DATA_BLOCK "DB_IN"	// DB 111
AUTHOR : M.Kögel
VERSION : 0.1
  STRUCT
   EMX_SPINDLE_RUN : BOOL ;	//Spindel läuft
   EMX_PROGRAM_RUN : BOOL ;	//Programm läuft
   EMX_FEED_HOLD : BOOL ;	//Vorschuboverride = 0 oder Voschub Stopp
   EMX_WARNING : BOOL ;	//Warnmeldung
   EMX_ERROR : BOOL ;	//Fehlermeldung
   EMX_FUNCTION_M20 : BOOL ;	//Funktion M20/M190
   EMX_PROGRAM_HALT : BOOL ;	//programmierter Halt "M00"
   EMX_AXIS_MOVE : BOOL ;	//mindestens eine Hauptachse in Bewegung
   EMX_MANUAL_MODE : BOOL ;	//Betriebsart Manuell
   EMX_TEACH_MODE : BOOL ;	//Betriebsart Teach
   EMX_SINGLE_MODE : BOOL ;	//Betriebsart Einzelsatz
   EMX_AUTO_MODE : BOOL ;	//Betriebsart Auto
   EMX_CYCLE_START : BOOL ;	//Zyklus Start (Starttaste - grün)
   EMX_MACHINE_ON : BOOL ;	//Maschine ist eingeschaltet (KEIN Not-Aus)
   EMX_NC_READY2RUN : BOOL ;	//NC-Betriebsbereit
   EMX_PROGRAM_END : BOOL ;	//Programm Ende
   EMB_PALLET_NUMBER : BYTE ;	//Nummer der Palette im Arbeitsraum
   EMX_PC_ACTIVE : BOOL ;	//Palettenwechsel aktiv
   EMX_SUS_DOOR_LOCKED : BOOL ;	//Rüstplatztüre(n) geschlossen und verriegelt
   EMX_PALLET_ON_SUS : BOOL ;	//Palette am Rüstplatz vorhanden
   EMX_ERROR_PULSE : BOOL ;	//Impuls von 1sec bei jeder Fehlermeldung
   EMX_PC_RELEASED : BOOL ;	//Freigabe für Palettenwechsel ist aktiv
   EMX_PC_PROCESS_END : BOOL ;	//Palettenwechsel beendet (nachdem Palette geklemmt)
   EMX_SUS_DOOR_CLOSED : BOOL ;	//Rüstplatztüre(n) geschlossen
   EMX_PC_CHANGE_POS : BOOL ;	//Maschinenpalette auf Übergabeposition (vor Hubbewegung)
   EMX_COOLANT_M8 : BOOL ;	//äußere Kühlschmierstoffzufuhr
   EMX_COOLANT_M7 : BOOL ;	//innere Kühlschmierstoffzufuhr
   EMX_FLUSH_PALLET : BOOL ;	//Spülung Palettenträger aktiv
   EMX_COOLANT_BACKFLOW : BOOL ;	//Förderpumpe Sammelbehälter (Rückförderung aus Maschine)
   EMX_COOLANT_LACK : BOOL ;	//Vorwarnung Kühlschmierstoffmangel
   EMX_COOLANT_MINLEVEL : BOOL ;	//Kühlschmierstoffanlage Füllstand minimum
   EMX_LUBRICAT_MINLEVEL : BOOL ;	//Zentralschmierung Füllstand minimum
   EMX_MQL_MINLEVEL : BOOL ;	//Minimalmengenschmierung Füllstand minimum
   EMX_HYDR_MINLEVEL : BOOL ;	//Hydraulikaggregat Werkzeugmaschine Füllstand minimum
   EMX_HYDRCHUCK_MINLEVEL : BOOL ;	//Hydraulikaggregat Spannhydraulik Füllstand minimum
   frei52 : BOOL ;
   frei53 : BOOL ;
   frei54 : BOOL ;
   frei55 : BOOL ;
   frei56 : BOOL ;
   frei57 : BOOL ;
   EMX_FEEDRATE_X : BOOL ;	//Vorschuboverride größer Wert "X"
   EMX_TOOL_LIFE : BOOL ;	//Standzeit des aktuellen Werkzeuges abgelaufen
   EMX_TOOL_CHANGE : BOOL ;	//Werkzeugwechsel aktiv
   EMX_MQL_ACTIVE : BOOL ;	//Minimalmengenschmierung aktiv (M34/M35)
   EMX_TOOL_LIFE_PREWARN : BOOL ;	//Die Standzeit des aktuellen Werkzeuges hat die Vorwarngrenze überschritten
   EMX_MAINTENANCE_REMIN : BOOL ;	//Wartungsaufruf (gemäß Betriebsanleitung; bei Maschinenfunktion (Dauer =250h)
   EMX_LUBRICAT_ACTIVE : BOOL ;	//High-Pegel, wenn die Zentral- (Maschinen)schmierung aktiviert ist
   ImxToolBreakage : BOOL ;	//Werkzeugbruch, welcher ein Stop auslöst
   EMX_ALARM_RESET : BOOL ;	//Meldung quittieren
   EMX_WORKROOM_DOOR : BOOL ;	//Arbeitsraumtüre(n) der Werkzeugmaschine geschlossen und verriegelt
   EMX_ZPS_RELEASE_EXT : BOOL ;	//Nullpunktspannsystem lösen (von extern)
   EMX_FIXTURE_ON_SUS : BOOL ;	//Palette mit (externem) Spannsystem auf Rüstplatz (MAS, RS4)
   frei74 : BOOL ;
   EMX_UNLOCK_FIXTURE : BOOL ;	//Freigabe für Spannvorrichtung lösen (Handling)
   frei76 : BOOL ;
   frei77 : BOOL ;
   EMX_OPERATING_MODE2 : BOOL ;	//Betriebsart_2 aktiv (Einrichtbetrieb)
   EMX_OPERATING_MODE3 : BOOL ;	//Betriebsart_3 aktiv (manueller Eingriff)
   EMX_OPERATING_MODE4 : BOOL ;	//Betriebsart_4 aktiv (erweiterter manueller Eingriff )
   EMX_AXIS_STANDSTILL : BOOL ;	//Achsenstillstand (Arbeitsraum) X/Y/Z/S/A/B/C-Achse
   EMX_STROBE_FUNCTION1 : BOOL ;	//Zustandswechsel an Funktionsaufruf (EMW_FUNCTION1)
   EMX_TURNTABLE_RUN : BOOL ;	//Fräs-Drehtisch läuft im Drehbetrieb
   frei86 : BOOL ;
   frei87 : BOOL ;
   EMX_SUS_PRESSURELESS : BOOL ;	//Medienübergabe am Rüstplatz (des PW oder des Rundspeichers) drucklos
   EMX_SUS_COUPLED : BOOL ;	//Andockeinheit (Medienversorgung) am Rüstplatz ausgefahren (gekuppelt)
   EMX_SUS_DOOR_OPENED : BOOL ;	//Rüstplatztüre des Speichersystem (z.B. RS4) vollständig geöffnet
   ImxOpenSusDoor : BOOL ;	//Rüstplatztüre(n) öffnen
   ImxCloseSusDoor : BOOL ;	//Rüstplatztüre(n) schließen
   frei95 : BOOL ;
   frei96 : BOOL ;
   frei97 : BOOL ;
   EMW_PARAMETER_1 : WORD ;	//Konfiguration über Maschinenparameter_1
   EMW_PARAMETER_2 : WORD ;	//Konfiguration über Maschinenparameter_2
   EMW_PARAMETER_3 : WORD ;	//Konfiguration über Maschinenparameter_3
   EMW_PARAMETER_4 : WORD ;	//Konfiguration über Maschinenparameter_4
   EMB_FEEDRATE : BYTE ;	//Stellung(Position) des Vorschubpotentiometers(Override)
   EMB_RAPID_VELOCITY : BYTE ;	//Stellung des Eilgangspotentiometers (Override)
   EMW_FUNCTION1 : WORD ;	//Funktionsaufruf durch Teileprogramm
   ImxDataRoutingBit0 : BOOL ;	//RANGIERER EINGANG BIT0
   ImxDataRoutingBit1 : BOOL ;	//RANGIERER EINGANG BIT1
   ImxDataRoutingBit2 : BOOL ;	//RANGIERER EINGANG BIT2
   ImxDataRoutingBit3 : BOOL ;	//RANGIERER EINGANG BIT3
   ImxDataRoutingBit4 : BOOL ;	//RANGIERER EINGANG BIT4
   ImxDataRoutingBit5 : BOOL ;	//RANGIERER EINGANG BIT5
   ImxDataRoutingBit6 : BOOL ;	//RANGIERER EINGANG BIT6
   ImxDataRoutingBit7 : BOOL ;	//RANGIERER EINGANG BIT7
   ImxDataRoutingBit8 : BOOL ;	//RANGIERER EINGANG BIT8
   ImxDataRoutingBit9 : BOOL ;	//RANGIERER EINGANG BIT9
   ImxDataRoutingBit10 : BOOL ;	//RANGIERER EINGANG BIT10
   ImxDataRoutingBit11 : BOOL ;	//RANGIERER EINGANG BIT11
   ImxDataRoutingBit12 : BOOL ;	//RANGIERER EINGANG BIT12
   ImxDataRoutingBit13 : BOOL ;	//RANGIERER EINGANG BIT13
   ImxDataRoutingBit14 : BOOL ;	//RANGIERER EINGANG BIT14
   ImxDataRoutingBit15 : BOOL ;	//RANGIERER EINGANG BIT15
   ImbSpindleOverride : BYTE ;	//Stellung des Spindeldrehzahlkorrekturschalters
  END_STRUCT ;	
BEGIN
END_DATA_BLOCK

DATA_BLOCK "DB_OUT"	// DB 112
AUTHOR : APetz
VERSION : 0.1
  STRUCT
   AMX_FEED_STOP : BOOL ;	//Vorschub Stopp  (mit Fehlermeldung)
   AMX_FEED_HOLD_CYCLE : BOOL ;	//Vorschub Halt (gilt nicht bei Eilgang-G00) mit Warnung
   AMX_SPINDLE_FEED_STOP : BOOL ;	//Spindel und Vorschub Stopp (mit Fehlermeldung)
   AMX_SPINDLE_FEED_STOP_P : BOOL ;	//Spindel und Vorschub Stopp nach abgearbeitetem Satz (mit Fehlermeldung)
   AMX_EMERGENCY_STOP : BOOL ;	//Not-Aus
   AMX_EMERGENCY_STOP_P : BOOL ;	//Not-Aus nach abgearbeitetem Satz
   AMX_LUBRICATION_LEVEL : BOOL ;	//Füllstandsüberwachung Schmieraggregat -> Warnmeldung
   AMX_SPINDLE_FEED_STOP_G0 : BOOL ;	//Spindel und Vorschub Stopp beim nächstem G0
   AMX_PC_RELEASE : BOOL ;	//Freigabe Palettenwechsler (Taste)
   AMX_PC_LOCK : BOOL ;	//Palettenwechsler sperren
   AMX_PC_ENABLE : BOOL ;	//Palettenwechselablauf freigeben
   AMX_STACKER_LOCK : BOOL ;	//Fahraufträge des Speichersystems vom und zum Rüstplatz sperren
   frei14 : BOOL ;
   frei15 : BOOL ;
   frei16 : BOOL ;
   frei17 : BOOL ;
   AMX_ERROR_KSS : BOOL ;	//Fehlermeldung Späneförderer/Kühlmittel
   AMX_FLOW_CONTROL_M7 : BOOL ;	//Kühlmitteldurchfluss im Kühlschmierstoff-Hochdruckkreis vorhanden
   AMX_FLOW_CONTROL_M8 : BOOL ;	//Kühlmitteldurchfluss im Kühlschmierstoff-Niederdruckkreis vorhanden
   frei23 : BOOL ;
   frei24 : BOOL ;
   frei25 : BOOL ;
   frei26 : BOOL ;
   frei27 : BOOL ;
   frei30 : BOOL ;
   frei31 : BOOL ;
   frei32 : BOOL ;
   frei33 : BOOL ;
   frei34 : BOOL ;
   frei35 : BOOL ;
   frei36 : BOOL ;
   frei37 : BOOL ;
   AMX_ZPS_RELEASED : BOOL ;	//Nullpunktspannsystem gelöst
   AMX_ZPS_CLAMPED : BOOL ;	//Nullpunktspannsystem gespannt/Verriegelt
   frei42 : BOOL ;
   frei43 : BOOL ;
   frei44 : BOOL ;
   frei45 : BOOL ;
   frei46 : BOOL ;
   frei47 : BOOL ;
   AMX_SUS_COUPLE : BOOL ;	//Hubzylinder für Andockeinheit (Medienversorgung) am Rüstplatz ausfahren
   frei51 : BOOL ;
   frei52 : BOOL ;
   frei53 : BOOL ;
   frei54 : BOOL ;
   frei55 : BOOL ;
   frei56 : BOOL ;
   frei57 : BOOL ;
   AMX_LOCK_NCSTART : BOOL ;	//Blockierung für NC-Start
   AMX_QUIT_FUNCTION1 : BOOL ;	//Quittierung des „Funktionsaufrufes aus Teileprogramm"
   AMX_QUIT_MTH : BOOL ;	//Rückmeldung von M-Funktion(en)
   frei63 : BOOL ;
   frei64 : BOOL ;
   frei65 : BOOL ;
   frei66 : BOOL ;
   frei67 : BOOL ;
   AMX_AXIS_MOVE_BACK : BOOL ;	//Rückzug in Werkzeugrichtung mit anschließendem Spindel- und Vorschub Halt
   frei71 : BOOL ;
   frei72 : BOOL ;
   frei73 : BOOL ;
   frei74 : BOOL ;
   frei75 : BOOL ;
   frei76 : BOOL ;
   frei77 : BOOL ;
   AMW_MESSAGENUMBER : INT ;	//Meldungsnummer aus Sonderoption
   AW_18 : WORD ;
  END_STRUCT ;	
BEGIN
END_DATA_BLOCK

ORGANIZATION_BLOCK "CYCL_EXC"	// OB 1
TITLE = "Main Program Sweep (Cycle)"
AUTHOR : APetz
VERSION : 0.1
VAR_TEMP
  OB1_EV_CLASS : BYTE ;	//Bits 0-3 = 1 (Coming event), Bits 4-7 = 1 (Event class 1)
  OB1_SCAN_1 : BYTE ;	//1 (Cold restart scan 1 of OB 1), 3 (Scan 2-n of OB 1)
  OB1_PRIORITY : BYTE ;	//Priority of OB Execution
  OB1_OB_NUMBR : BYTE ;	//1 (Organization block 1, OB1)
  OB1_RESERVED_1 : BYTE ;	//Reserved for system
  OB1_RESERVED_2 : BYTE ;	//Reserved for system
  OB1_PREV_CYCLE : INT ;	//Cycle time of previous OB1 scan (milliseconds)
  OB1_MIN_CYCLE : INT ;	//Minimum cycle time of OB1 (milliseconds)
  OB1_MAX_CYCLE : INT ;	//Maximum cycle time of OB1 (milliseconds)
  OB1_DATE_TIME : DATE_AND_TIME ;	//Date and time OB1 started
END_VAR
BEGIN
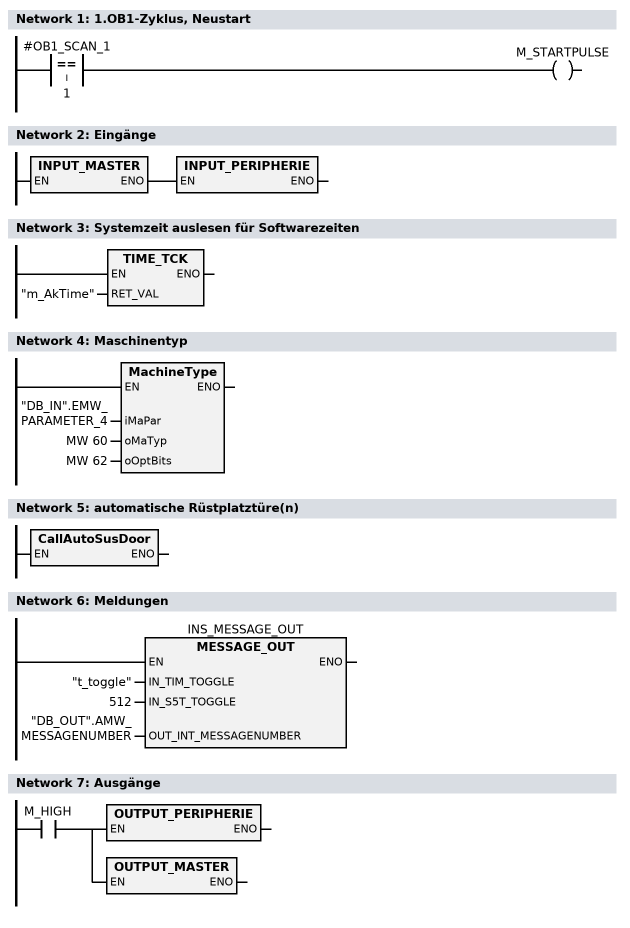
NETWORK
TITLE = 1.OB1-Zyklus, Neustart
//bilden eines Startimpulses
//OB1_SCAN_1
//Wert B#16#01 bedeutet: Abschluß des Neustarts (Warmstarts)·
      L     #OB1_SCAN_1;
      L     1;
      ==I;
      =     "M_STARTPULSE";
NETWORK
TITLE = Eingänge
//Eingänge von Mastersystem einlesen
//Eingänge von Peripherie lesen
      A(;
      CALL  "INPUT_MASTER";
      A     BR;
      );
      JNB   _001;
      CALL  "INPUT_PERIPHERIE";
_001: NOP   0;
NETWORK
TITLE = Systemzeit auslesen für Softwarezeiten
      CALL  "TIME_TCK" (
           RET_VAL                  := "m_AkTime");
      NOP   0;
NETWORK
TITLE = Maschinentyp
      CALL  "MachineType" (
           iMaPar                   := "DB_IN".EMW_PARAMETER_4,
           oMaTyp                   := MW 60,
           oOptBits                 := MW 62);
      NOP   0;
NETWORK
TITLE = automatische Rüstplatztüre(n)
      CALL  "CallAutoSusDoor";
      NOP   0;
NETWORK
TITLE = Meldungen
//Übergabe der Meldungen zum Master
//Wenn mehrere Meldungen anstehen, werden diese durchgetaktet
      CALL  "MESSAGE_OUT" , "INS_MESSAGE_OUT" (
           IN_TIM_TOGGLE            := "t_toggle",
           IN_S5T_TOGGLE            := 512,
           OUT_INT_MESSAGENUMBER    := "DB_OUT".AMW_MESSAGENUMBER);
      NOP   0;
NETWORK
TITLE = Ausgänge
//Ausgänge Peripherie schreiben
//Ausgänge an Mastersystem schreiben
      A     "M_HIGH";
      =     L 20.0;
      A     L 20.0;
      JNB   _002;
      CALL  "OUTPUT_PERIPHERIE";
_002: NOP   0;
      A     L 20.0;
      JNB   _003;
      CALL  "OUTPUT_MASTER";
_003: NOP   0;
END_ORGANIZATION_BLOCK

ORGANIZATION_BLOCK "I/O_FLT1"	// OB 82
TITLE = "I/O Point Fault"
VERSION : 0.1
VAR_TEMP
  OB82_EV_CLASS : BYTE ;	//16#39, Event class 3, Entering event state, Internal fault event
  OB82_FLT_ID : BYTE ;	//16#XX, Fault identifcation code
  OB82_PRIORITY : BYTE ;	//Priority of OB Execution
  OB82_OB_NUMBR : BYTE ;	//82 (Organization block 82, OB82)
  OB82_RESERVED_1 : BYTE ;	//Reserved for system
  OB82_IO_FLAG : BYTE ;	//Input (01010100), Output (01010101)
  OB82_MDL_ADDR : INT ;	//Base address of module with fault
  OB82_MDL_DEFECT : BOOL ;	//Module defective
  OB82_INT_FAULT : BOOL ;	//Internal fault
  OB82_EXT_FAULT : BOOL ;	//External fault
  OB82_PNT_INFO : BOOL ;	//Point information
  OB82_EXT_VOLTAGE : BOOL ;	//External voltage low
  OB82_FLD_CONNCTR : BOOL ;	//Field wiring connector missing
  OB82_NO_CONFIG : BOOL ;	//Module has no configuration data
  OB82_CONFIG_ERR : BOOL ;	//Module has configuration error
  OB82_MDL_TYPE : BYTE ;	//Type of module
  OB82_SUB_NDL_ERR : BOOL ;	//Sub-Module is missing or has error
  OB82_COMM_FAULT : BOOL ;	//Communication fault
  OB82_MDL_STOP : BOOL ;	//Module is stopped
  OB82_WTCH_DOG_FLT : BOOL ;	//Watch dog timer stopped module
  OB82_INT_PS_FLT : BOOL ;	//Internal power supply fault
  OB82_PRIM_BATT_FLT : BOOL ;	//Primary battery is in fault
  OB82_BCKUP_BATT_FLT : BOOL ;	//Backup battery is in fault
  OB82_RESERVED_2 : BOOL ;	//Reserved for system
  OB82_RACK_FLT : BOOL ;	//Rack fault, only for bus interface module
  OB82_PROC_FLT : BOOL ;	//Processor fault
  OB82_EPROM_FLT : BOOL ;	//EPROM fault
  OB82_RAM_FLT : BOOL ;	//RAM fault
  OB82_ADU_FLT : BOOL ;	//ADU fault
  OB82_FUSE_FLT : BOOL ;	//Fuse fault
  OB82_HW_INTR_FLT : BOOL ;	//Hardware interupt input in fault
  OB82_RESERVED_3 : BOOL ;	//Reserved for system
  OB82_DATE_TIME : DATE_AND_TIME ;	//Date and time OB82 started
END_VAR
BEGIN
NETWORK
TITLE =
END_ORGANIZATION_BLOCK

ORGANIZATION_BLOCK "OBNL_FLT"	// OB 85
TITLE = "Organization Block (OB) Not Loaded Fault"
VERSION : 0.1
VAR_TEMP
  OB85_EV_CLASS : BYTE ;	//16#35 Event class 3
  OB85_FLT_ID : BYTE ;	//16#XX, Fault identification code
  OB85_PRIORITY : BYTE ;	//Priority of OB Execution
  OB85_OB_NUMBR : BYTE ;	//85 (Organization block 85, OB85)
  OB85_RESERVED_1 : BYTE ;	//Reserved for system
  OB85_RESERVED_2 : BYTE ;	//Reserved for system
  OB85_RESERVED_3 : INT ;	//Reserved for system
  OB85_ERR_EV_CLASS : BYTE ;	//Class of event causing error
  OB85_ERR_EV_NUM : BYTE ;	//Number of event causing error
  OB85_OB_PRIOR : BYTE ;	//Priority of OB causing error
  OB85_OB_NUM : BYTE ;	//Number of OB causing error
  OB85_DATE_TIME : DATE_AND_TIME ;	//Date and time OB85 started
END_VAR
BEGIN
NETWORK
TITLE =
END_ORGANIZATION_BLOCK

ORGANIZATION_BLOCK "RACK_FLT"	// OB 86
TITLE = "Loss Of Rack Fault"
VERSION : 0.1
VAR_TEMP
  OB86_EV_CLASS : BYTE ;	//16#38/39 Event class 3
  OB86_FLT_ID : BYTE ;	//16#C1/C4/C5, Fault identifcation code
  OB86_PRIORITY : BYTE ;	//Priority of OB Execution
  OB86_OB_NUMBR : BYTE ;	//86 (Organization block 86, OB86)
  OB86_RESERVED_1 : BYTE ;	//Reserved for system
  OB86_RESERVED_2 : BYTE ;	//Reserved for system
  OB86_MDL_ADDR : INT ;	//Base address of IM module in rack with fault
  OB86_RACKS_FLTD : ARRAY  [0 .. 31 ] OF BOOL ;	//Racks in fault
  OB86_DATE_TIME : DATE_AND_TIME ;	//Date and time OB86 started
END_VAR
BEGIN
NETWORK
TITLE =
END_ORGANIZATION_BLOCK

ORGANIZATION_BLOCK "START"	// OB 100
TITLE = "Complete Restart"
VERSION : 0.1
VAR_TEMP
  OB100_EV_CLASS : BYTE ;	//16#13, Event class 1, Entering event state, Event logged in diagnostic buffer
  OB100_STRTUP : BYTE ;	//16#81/82/83/84 Method of startup
  OB100_PRIORITY : BYTE ;	//Priority of OB Execution
  OB100_OB_NUMBR : BYTE ;	//100 (Organization block 100, OB100)
  OB100_RESERVED_1 : BYTE ;	//Reserved for system
  OB100_RESERVED_2 : BYTE ;	//Reserved for system
  OB100_STOP : WORD ;	//Event that caused CPU to stop (16#4xxx)
  OB100_STRT_INFO : DWORD ;	//Information on how system started
  OB100_DATE_TIME : DATE_AND_TIME ;	//Date and time OB100 started
END_VAR
BEGIN
NETWORK
TITLE = Merker als Konstanten EINMALIG festlegen
//Bei KOP/FUP kann True oder False nicht als Konstante übergeben werden. Deshalb 
//definieren wir hier jeweils einen Merker, der immer true ist und einen Merker, 
//der immer false ist.
//Das Resetbit wird am Ende des OB1 sofort wieder zurückgesetzt, damit das 
//Resetbit nur für EINEN Zyklus ansteht.
      SET;
      R     "M_LOW";
      S     "M_HIGH";
      S     "m_inbetriebnahme";
END_ORGANIZATION_BLOCK

ORGANIZATION_BLOCK "PROG_ERR"	// OB 121
TITLE = "Programming Error"
VERSION : 0.1
VAR_TEMP
  OB121_EV_CLASS : BYTE ;	//16#25, Event class 2, Entering event state, Internal fault event
  OB121_SW_FLT : BYTE ;	//16#XX Software programming fault
  OB121_PRIORITY : BYTE ;	//Priority of OB Execution
  OB121_OB_NUMBR : BYTE ;	//121 (Organization block 121, OB121)
  OB121_BLK_TYPE : BYTE ;	//16#88/8A/8B/8C/8E Type of block fault occured in
  OB121_RESERVED_1 : BYTE ;	//Reserved for system
  OB121_FLT_REG : WORD ;	//16#XX Specific register that caused fault
  OB121_BLK_NUM : WORD ;	//Number of block that programming fault occured in
  OB121_PRG_ADDR : WORD ;	//Address in block where programming fault occured
  OB121_DATE_TIME : DATE_AND_TIME ;	//Date and time OB121 started
END_VAR
BEGIN
// (block stored without names or comments; labels and parameter names are numbered)
END_ORGANIZATION_BLOCK

ORGANIZATION_BLOCK "MOD_ERR"	// OB 122
TITLE = "Module Access Error"
VERSION : 0.1
VAR_TEMP
  OB122_EV_CLASS : BYTE ;	//16#29, Event class 2, Entering event state, Internal fault event
  OB122_SW_FLT : BYTE ;	//16#XX Software error code
  OB122_PRIORITY : BYTE ;	//Priority of OB Execution
  OB122_OB_NUMBR : BYTE ;	//122 (Organization block 122, OB122)
  OB122_BLK_TYPE : BYTE ;	//16#88/8C/8E Type of block fault occured in
  OB122_MEM_AREA : BYTE ;	//Memory area where access error occured
  OB122_MEM_ADDR : WORD ;	//Memory address where access error occured
  OB122_BLK_NUM : WORD ;	//Block number in which error occured
  OB122_PRG_ADDR : WORD ;	//Program address where error occured
  OB122_DATE_TIME : DATE_AND_TIME ;	//Date and time OB1 started
END_VAR
BEGIN
// (block stored without names or comments; labels and parameter names are numbered)
END_ORGANIZATION_BLOCK

FUNCTION_BLOCK FB 20
AUTHOR : SPAC_slh
FAMILY : AUTOMAT
NAME : SusDoor
VERSION : 0.1
BEGIN
// (block stored without names or comments; labels and parameter names are numbered)
NETWORK
TITLE =
      A     DB111.DBX 1.5;
      =     L 11.2;
NETWORK
TITLE =
      L     DIB 0;
      AW    W#16#F;
      TAR1  LD 0;
      LAR1  P#L 8.0;
      L     B#16#0;
      T     LW [AR1,P#0.0];
      TAK;
      +AR1;
      A     M 0.1;
      S     L [AR1,P#0.0];
      LAR1  LD 0;
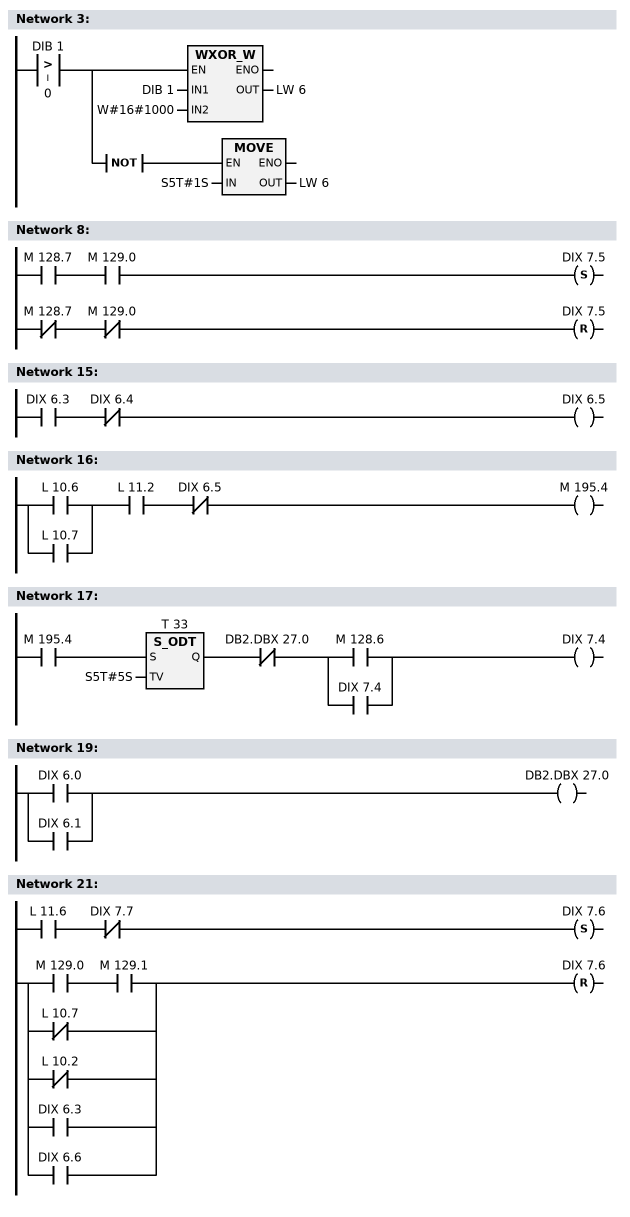
NETWORK
TITLE =
      L     DIB 1;
      L     0;
      >I;
      =     L 13.0;
      A     L 13.0;
      JNB   M001;
      L     DIB 1;
      L     W#16#1000;
      XOW;
      T     LW 6;
M001: NOP   0;
      A     L 13.0;
      NOT;
      JNB   M002;
      L     S5T#1S;
      T     LW 6;
M002: NOP   0;
NETWORK
TITLE =
      A     L 8.1;
      =     L 10.6;
NETWORK
TITLE =
      O     L 8.2;
      O     L 8.3;
      O     L 8.4;
      O     L 8.5;
      =     L 10.7;
NETWORK
TITLE =
      O     L 8.3;
      O     L 8.5;
      =     L 10.3;
NETWORK
TITLE =
      O     L 8.4;
      O     L 8.5;
      =     L 10.4;
NETWORK
TITLE =
      A     M 128.7;
      A     M 129.0;
      S     DIX 7.5;
      AN    M 128.7;
      AN    M 129.0;
      R     DIX 7.5;
      NOP   0;
NETWORK
TITLE =
      A     M 129.1;
      AN    DIX 7.5;
      A     M 128.7;
      AN    M 129.0;
      =     L 11.6;
NETWORK
TITLE =
      A     M 129.1;
      AN    DIX 7.5;
      AN    M 128.7;
      A     M 129.0;
      =     L 11.7;
NETWORK
TITLE =
      A(;
      O     L 8.2;
      O     L 8.4;
      );
      AN    M 129.1;
      =     L 10.1;
      A     L 10.1;
      A     DB111.DBX 9.4;
      AN    DB111.DBX 9.3;
      =     L 12.0;
NETWORK
TITLE =
      A     L 10.1;
      AN    DB111.DBX 9.4;
      A     DB111.DBX 9.3;
      =     L 12.1;
NETWORK
TITLE =
      L     0;
      L     DB2.DBW 27;
      <>I;
      =     L 11.5;
NETWORK
TITLE =
      A     M 129.5;
      A(;
      O     M 129.6;
      O     DIX 2.0;
      );
      =     L 10.5;
NETWORK
TITLE =
      A     DIX 6.3;
      AN    DIX 6.4;
      =     DIX 6.5;
NETWORK
TITLE =
      A(;
      O     L 10.6;
      O     L 10.7;
      );
      A     L 11.2;
      AN    DIX 6.5;
      =     M 195.4;
NETWORK
TITLE =
      A(;
      A     M 195.4;
      L     S5T#5S;
      SD    T 33;
      NOP   0;
      NOP   0;
      NOP   0;
      A     T 33;
      );
      AN    DB2.DBX 27.0;
      A(;
      O     M 128.6;
      O     DIX 7.4;
      );
      =     DIX 7.4;
NETWORK
TITLE =
      A     M 128.6;
      =     L 14.0;
      BLD   103;
      A     M 195.4;
      =     L 14.1;
      BLD   103;
      A     DB111.DBX 7.0;
      =     L 14.2;
      BLD   103;
      AN    L 10.6;
      JNB   M003;
      BLD   1;
      L     W#16#1002;
      T     LW 15;
      L     14;
      T     LW 17;
      L     101;
      T     LW 19;
      L     P#DBX 56.0;
      T     LD 21;
      L     L#3000;
      T     LD 25;
      L     L#3000;
      T     LD 29;
      L     L#500;
      T     LD 33;
      A     DIX 6.0;
      =     L 37.0;
      A     DIX 6.1;
      =     L 37.1;
      A     DB2.DBX 27.1;
      =     L 37.2;
      UC    FC 102;
      {     P#L 15.0, P#M 12.0, P#L 25.0, P#L 29.0, P#L 33.0, P#L 14.0, P#L 14.1, P#L 14.2, P#L 37.0, P#L 37.1, P#L 37.2 };
      A     L 37.0;
      =     DIX 6.0;
      A     L 37.1;
      =     DIX 6.1;
      A     L 37.2;
      =     DB2.DBX 27.1;
      BLD   2;
M003: NOP   0;
NETWORK
TITLE =
      O     DIX 6.0;
      O     DIX 6.1;
      =     DB2.DBX 27.0;
NETWORK
TITLE =
      A     DIX 7.4;
      AN    L 11.5;
      AN    DIX 6.5;
      =     L 10.2;
NETWORK
TITLE =
      A     L 11.6;
      AN    DIX 7.7;
      S     DIX 7.6;
      A(;
      A     M 129.0;
      A     M 129.1;
      ON    L 10.7;
      ON    L 10.2;
      O     DIX 6.3;
      O     DIX 6.6;
      );
      R     DIX 7.6;
      NOP   0;
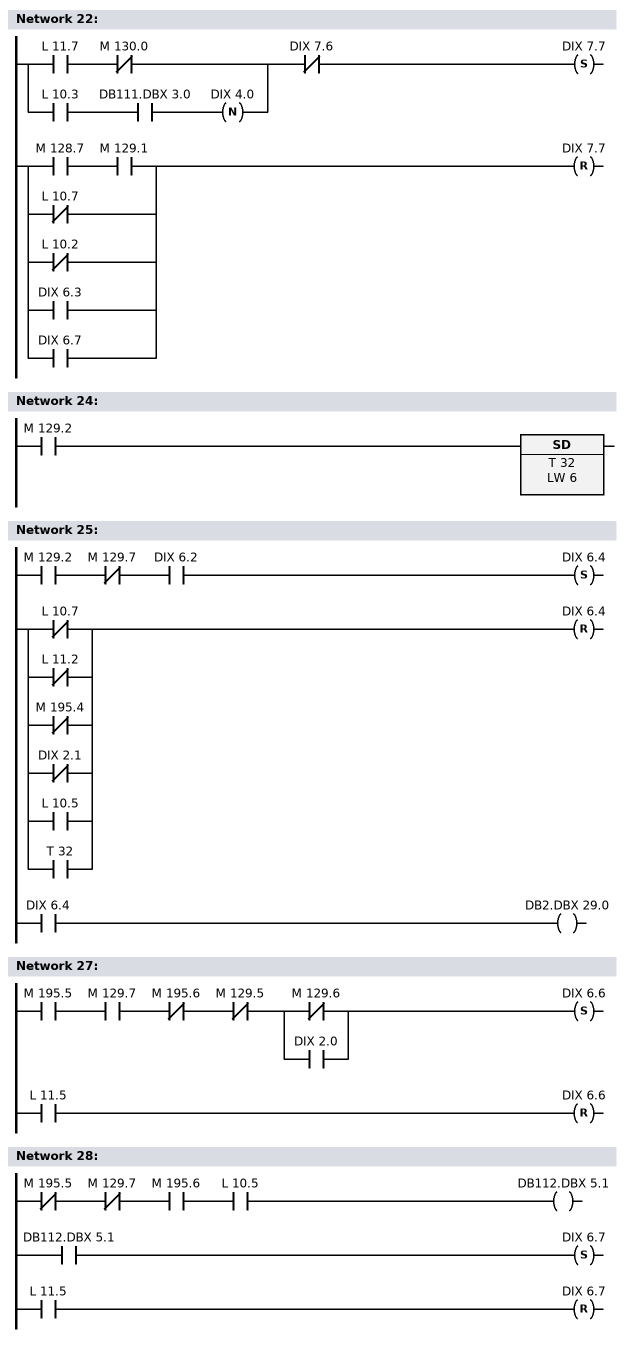
NETWORK
TITLE =
      A(;
      A     L 11.7;
      AN    M 130.0;
      O(;
      A     L 10.3;
      A     DB111.DBX 3.0;
      FN    DIX 4.0;
      );
      );
      AN    DIX 7.6;
      S     DIX 7.7;
      A(;
      A     M 128.7;
      A     M 129.1;
      ON    L 10.7;
      ON    L 10.2;
      O     DIX 6.3;
      O     DIX 6.7;
      );
      R     DIX 7.7;
      NOP   0;
NETWORK
TITLE =
      A(;
      A     DB111.DBX 7.0;
      R     DIX 6.3;
      A     M 129.2;
      AN    M 129.7;
      S     DIX 6.3;
      A     DIX 6.3;
      );
      AN    DB2.DBX 29.0;
      =     DB2.DBX 29.1;
NETWORK
TITLE =
      A     M 129.2;
      L     LW 6;
      SD    T 32;
NETWORK
TITLE =
      A     M 129.2;
      AN    M 129.7;
      A     DIX 6.2;
      S     DIX 6.4;
      A(;
      ON    L 10.7;
      ON    L 11.2;
      ON    M 195.4;
      ON    DIX 2.1;
      O     L 10.5;
      O     T 32;
      );
      R     DIX 6.4;
      A     DIX 6.4;
      =     DB2.DBX 29.0;
NETWORK
TITLE =
      A     L 10.2;
      =     L 14.0;
      A     L 14.0;
      AN    DIX 6.4;
      =     L 11.3;
      A     L 14.0;
      A(;
      A     L 11.3;
      A(;
      A     L 10.7;
      A(;
      O     DIX 7.6;
      O     L 12.0;
      );
      O;
      A     L 10.6;
      A     L 11.6;
      );
      O     DIX 6.6;
      );
      =     M 195.5;
      R     DIX 6.7;
      A     L 14.0;
      AN    M 130.0;
      =     L 11.4;
      A     L 14.0;
      A(;
      A     L 11.4;
      A(;
      A     L 10.7;
      A(;
      O     DIX 7.7;
      O     DIX 6.4;
      O     L 12.1;
      );
      O;
      A     L 10.6;
      A     L 11.7;
      );
      O     DIX 6.7;
      );
      =     M 195.6;
      R     DIX 6.6;
NETWORK
TITLE =
      A     M 195.5;
      A     M 129.7;
      AN    M 195.6;
      AN    M 129.5;
      A(;
      ON    M 129.6;
      O     DIX 2.0;
      );
      S     DIX 6.6;
      A     L 11.5;
      R     DIX 6.6;
      NOP   0;
NETWORK
TITLE =
      AN    M 195.5;
      AN    M 129.7;
      A     M 195.6;
      A     L 10.5;
      =     DB112.DBX 5.1;
      A     DB112.DBX 5.1;
      S     DIX 6.7;
      A     L 11.5;
      R     DIX 6.7;
      NOP   0;
NETWORK
TITLE =
      A     M 129.5;
      =     L 14.0;
      BLD   103;
      A     M 195.6;
      =     L 14.1;
      BLD   103;
      A     M 129.7;
      =     L 14.2;
      BLD   103;
      A     M 195.5;
      =     L 14.3;
      BLD   103;
      A     M 0.0;
      =     L 14.4;
      BLD   103;
      A     DB111.DBX 7.0;
      =     L 14.5;
      BLD   103;
      A     M 0.0;
      =     L 14.6;
      BLD   103;
      A     M 0.0;
      =     L 14.7;
      BLD   103;
      A     M 0.0;
      =     L 15.0;
      BLD   103;
      AN    L 10.6;
      JNB   M004;
      BLD   1;
      L     W#16#1002;
      T     LW 16;
      L     14;
      T     LW 18;
      L     101;
      T     LW 20;
      L     P#DBX 70.0;
      T     LD 22;
      L     L#100;
      T     LD 26;
      L     L#7000;
      T     LD 30;
      L     L#1000;
      T     LD 34;
      A     DB2.DBX 92.0;
      =     L 38.0;
      A     DB2.DBX 92.1;
      =     L 38.1;
      A     DB2.DBX 27.2;
      =     L 38.2;
      A     DB2.DBX 27.3;
      =     L 38.3;
      A     DB2.DBX 27.4;
      =     L 38.4;
      UC    FC 101;
      {     P#L 16.0, P#M 12.0, P#L 26.0, P#L 30.0, P#L 34.0, P#L 14.0, P#L 14.1, P#L 14.2, P#L 14.3, P#L 14.4, P#L 14.5, P#L 14.6, P#L 14.7, P#L 15.0, P#L 38.0, P#L 38.1, P#L 38.2, P#L 38.3, P#L 38.4 };
      A     L 38.0;
      =     DB2.DBX 92.0;
      A     L 38.1;
      =     DB2.DBX 92.1;
      A     L 38.2;
      =     DB2.DBX 27.2;
      A     L 38.3;
      =     DB2.DBX 27.3;
      A     L 38.4;
      =     DB2.DBX 27.4;
      BLD   2;
M004: NOP   0;
NETWORK
TITLE =
      A     M 129.6;
      =     L 14.0;
      BLD   103;
      A     M 195.6;
      =     L 14.1;
      BLD   103;
      A     M 129.7;
      =     L 14.2;
      BLD   103;
      A     M 195.5;
      =     L 14.3;
      BLD   103;
      A     M 0.0;
      =     L 14.4;
      BLD   103;
      A     DB111.DBX 7.0;
      =     L 14.5;
      BLD   103;
      A     M 0.0;
      =     L 14.6;
      BLD   103;
      A     M 0.0;
      =     L 14.7;
      BLD   103;
      A     M 0.0;
      =     L 15.0;
      BLD   103;
      AN    L 10.6;
      AN    DIX 2.0;
      JNB   M005;
      BLD   1;
      L     W#16#1002;
      T     LW 16;
      L     14;
      T     LW 18;
      L     101;
      T     LW 20;
      L     P#DBX 84.0;
      T     LD 22;
      L     L#100;
      T     LD 26;
      L     L#7000;
      T     LD 30;
      L     L#1000;
      T     LD 34;
      A     DB2.DBX 92.2;
      =     L 38.0;
      A     DB2.DBX 92.3;
      =     L 38.1;
      A     DB2.DBX 27.5;
      =     L 38.2;
      A     DB2.DBX 27.6;
      =     L 38.3;
      A     DB2.DBX 27.7;
      =     L 38.4;
      UC    FC 101;
      {     P#L 16.0, P#M 12.0, P#L 26.0, P#L 30.0, P#L 34.0, P#L 14.0, P#L 14.1, P#L 14.2, P#L 14.3, P#L 14.4, P#L 14.5, P#L 14.6, P#L 14.7, P#L 15.0, P#L 38.0, P#L 38.1, P#L 38.2, P#L 38.3, P#L 38.4 };
      A     L 38.0;
      =     DB2.DBX 92.2;
      A     L 38.1;
      =     DB2.DBX 92.3;
      A     L 38.2;
      =     DB2.DBX 27.5;
      A     L 38.3;
      =     DB2.DBX 27.6;
      A     L 38.4;
      =     DB2.DBX 27.7;
      BLD   2;
M005: NOP   0;
NETWORK
TITLE =
      A     M 129.3;
      =     L 14.0;
      BLD   103;
      A     M 195.6;
      =     L 14.1;
      BLD   103;
      A     DB111.DBX 7.0;
      =     L 14.2;
      BLD   103;
      AN    L 10.6;
      JNB   M006;
      BLD   1;
      L     W#16#1002;
      T     LW 15;
      L     14;
      T     LW 17;
      L     101;
      T     LW 19;
      L     P#DBX 98.0;
      T     LD 21;
      L     L#2000;
      T     LD 25;
      L     L#2000;
      T     LD 29;
      L     L#1500;
      T     LD 33;
      A     DIX 7.0;
      =     L 37.0;
      A     DIX 7.1;
      =     L 37.1;
      A     DB2.DBX 28.1;
      =     L 37.2;
      UC    FC 102;
      {     P#L 15.0, P#M 12.0, P#L 25.0, P#L 29.0, P#L 33.0, P#L 14.0, P#L 14.1, P#L 14.2, P#L 37.0, P#L 37.1, P#L 37.2 };
      A     L 37.0;
      =     DIX 7.0;
      A     L 37.1;
      =     DIX 7.1;
      A     L 37.2;
      =     DB2.DBX 28.1;
      BLD   2;
M006: NOP   0;
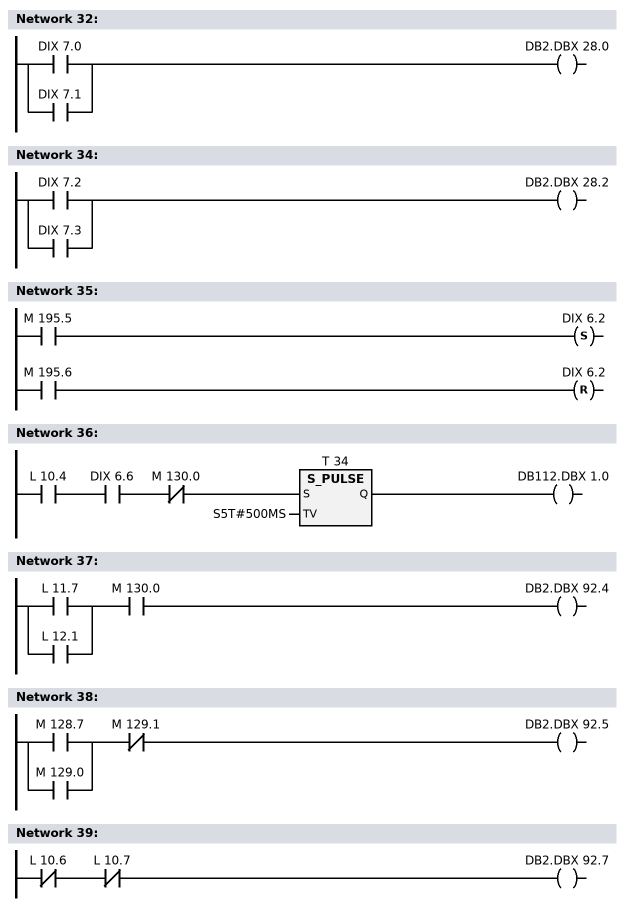
NETWORK
TITLE =
      O     DIX 7.0;
      O     DIX 7.1;
      =     DB2.DBX 28.0;
NETWORK
TITLE =
      A     M 129.4;
      =     L 14.0;
      BLD   103;
      A     M 195.5;
      =     L 14.1;
      BLD   103;
      A     DB111.DBX 7.0;
      =     L 14.2;
      BLD   103;
      AN    L 10.6;
      JNB   M007;
      BLD   1;
      L     W#16#1002;
      T     LW 15;
      L     14;
      T     LW 17;
      L     101;
      T     LW 19;
      L     P#DBX 112.0;
      T     LD 21;
      L     L#2000;
      T     LD 25;
      L     L#2000;
      T     LD 29;
      L     L#800;
      T     LD 33;
      A     DIX 7.2;
      =     L 37.0;
      A     DIX 7.3;
      =     L 37.1;
      A     DB2.DBX 28.3;
      =     L 37.2;
      UC    FC 102;
      {     P#L 15.0, P#M 12.0, P#L 25.0, P#L 29.0, P#L 33.0, P#L 14.0, P#L 14.1, P#L 14.2, P#L 37.0, P#L 37.1, P#L 37.2 };
      A     L 37.0;
      =     DIX 7.2;
      A     L 37.1;
      =     DIX 7.3;
      A     L 37.2;
      =     DB2.DBX 28.3;
      BLD   2;
M007: NOP   0;
NETWORK
TITLE =
      O     DIX 7.2;
      O     DIX 7.3;
      =     DB2.DBX 28.2;
NETWORK
TITLE =
      A     M 195.5;
      S     DIX 6.2;
      A     M 195.6;
      R     DIX 6.2;
      NOP   0;
NETWORK
TITLE =
      A     L 10.4;
      A     DIX 6.6;
      AN    M 130.0;
      L     S5T#500MS;
      SP    T 34;
      NOP   0;
      NOP   0;
      NOP   0;
      A     T 34;
      =     DB112.DBX 1.0;
NETWORK
TITLE =
      A(;
      O     L 11.7;
      O     L 12.1;
      );
      A     M 130.0;
      =     DB2.DBX 92.4;
NETWORK
TITLE =
      A(;
      O     M 128.7;
      O     M 129.0;
      );
      AN    M 129.1;
      =     DB2.DBX 92.5;
NETWORK
TITLE =
      AN    L 10.6;
      AN    L 10.7;
      =     DB2.DBX 92.7;
END_FUNCTION_BLOCK

FUNCTION_BLOCK FB 100
AUTHOR : SPAC_slh
NAME : MSG
VERSION : 0.1
BEGIN
// (block stored without names or comments; labels and parameter names are numbered)
NETWORK
TITLE =
      OPN   DB 2;
      L     0;
      T     DIW 518;
      TAR1  LD 0;
      LAR1  P#DIX 6.0;
      L     128;
M001: L     0;
      T     DID [AR1,P#0.0];
      +AR1  P#4.0;
      TAK;
      LOOP  M001;
NETWORK
TITLE =
      L     0;
M002: T     LW 4;
      SLW   4;
      LAR1;
      L     0;
      L     DBW [AR1,P#0.0];
      ==I;
      JC    M005;
      CAW;
M003: T     LW 8;
      DTR;
      SRD   23;
      +     -127;
      T     LB 12;
      L     LW 4;
      SLW   4;
      +I;
      +     1;
      LAR1  P#DIX 6.0;
      L     DIW 518;
      SLW   4;
      +AR1;
      TAK;
      T     DIW [AR1,P#0.0];
      L     255;
      L     DIW 518;
      >I;
      JCN   M004;
      +     1;
      T     DIW 518;
M004: L     0;
      LAR1  P#L 10.0;
      T     LW [AR1,P#0.0];
      L     LB 12;
      +AR1;
      S     L [AR1,P#0.0];
      L     LW 10;
      CAW;
      INVI;
      L     LW 8;
      AW;
      L     0;
      <>I;
      TAK;
      JC    M003;
M005: L     31;
      L     LW 4;
      +     1;
      >=I;
      JC    M002;
NETWORK
TITLE =
      L     0;
      L     DIW 6;
      <>I;
      JC    M010;
      L     32;
M006: T     LW 4;
      SLW   4;
      LAR1;
      L     0;
      L     DBW [AR1,P#0.0];
      ==I;
      JC    M009;
      CAW;
M007: T     LW 8;
      DTR;
      SRD   23;
      +     -127;
      T     LB 12;
      L     LW 4;
      SLW   4;
      +I;
      +     1;
      LAR1  P#DIX 6.0;
      L     DIW 518;
      SLW   4;
      +AR1;
      TAK;
      T     DIW [AR1,P#0.0];
      L     255;
      L     DIW 518;
      >I;
      JCN   M008;
      +     1;
      T     DIW 518;
M008: L     0;
      LAR1  P#L 10.0;
      T     LW [AR1,P#0.0];
      L     LB 12;
      +AR1;
      S     L [AR1,P#0.0];
      L     LW 10;
      CAW;
      INVI;
      L     LW 8;
      AW;
      L     0;
      <>I;
      TAK;
      JC    M007;
M009: L     63;
      L     LW 4;
      +     1;
      >=I;
      JC    M006;
M010: NOP   0;
NETWORK
TITLE =
      LAR1  LD 0;
      L     0;
      L     DIW 6;
      <>I;
      L     DIW 2;
      SD    T [DIW 0];
      JC    M011;
      L     0;
      T     DIW 520;
M011: AN    T [DIW 0];
      JC    M014;
      L     255;
      L     DIW 520;
      +     1;
      <I;
      JCN   M012;
      L     0;
M012: T     DIW 520;
      TAR1  LD 0;
      LAR1  P#DIX 6.0;
      L     DIW 520;
      SLW   4;
      +AR1;
      L     0;
      L     DIW [AR1,P#0.0];
      ==I;
      LAR1  LD 0;
      JCN   M013;
      L     0;
      T     DIW 520;
M013: CLR;
      L     DIW 2;
      SD    T [DIW 0];
      SET;
      SD    T [DIW 0];
M014: TAR1  LD 0;
      LAR1  P#DIX 6.0;
      L     DIW 520;
      SLW   4;
      +AR1;
      L     DIW [AR1,P#0.0];
      LAR1  LD 0;
      T     LW 6;
NETWORK
TITLE =
      L     LW 6;
      T     DIW 4;
END_FUNCTION_BLOCK

FUNCTION FC 90 : VOID
AUTHOR : APetz
FAMILY : GENERAL
NAME : General
VERSION : 1.0
BEGIN
// (block stored without names or comments; labels and parameter names are numbered)
NETWORK
TITLE =
      L     #PARAM1;
      DTB;
      T     LW 0;
      AW    W#16#F;
      T     #PARAM6;
      L     LW 0;
      AW    W#16#F0;
      SRW   4;
      T     #PARAM7;
      L     LW 0;
      AW    W#16#F00;
      SRW   8;
      T     #PARAM8;
      L     LW 0;
      AW    W#16#F000;
      SRW   12;
      T     #PARAM9;
      L     LW 0;
      AW    W#16#FF;
      BTI;
      T     #PARAM5;
      L     LW 0;
      CAW;
      AW    W#16#FF;
      BTI;
      T     #PARAM4;
      L     #PARAM2;
      JL    M001;
      JU    M002;
      JU    M003;
      JU    M004;
      JU    M005;
M001: CLR;
      JU    M007;
M002: L     #PARAM6;
      JU    M006;
M003: L     #PARAM7;
      JU    M006;
M004: L     #PARAM8;
      JU    M006;
M005: L     #PARAM9;
M006: L     #PARAM3;
      ==I;
M007: =     #PARAM10;
END_FUNCTION

FUNCTION FC 91 : VOID
AUTHOR : A.Petz
VERSION : 0.1
BEGIN
// (block stored without names or comments; labels and parameter names are numbered)
NETWORK
TITLE =
      L     #PARAM1;
      L     1;
      ==I;
      JCN   M001;
      L     #PARAM2;
      CAW;
      T     #PARAM3;
M001: NOP   0;
      SET;
      SAVE;
END_FUNCTION

FUNCTION FC 92 : VOID
AUTHOR : A.Petz
VERSION : 0.1
BEGIN
// (block stored without names or comments; labels and parameter names are numbered)
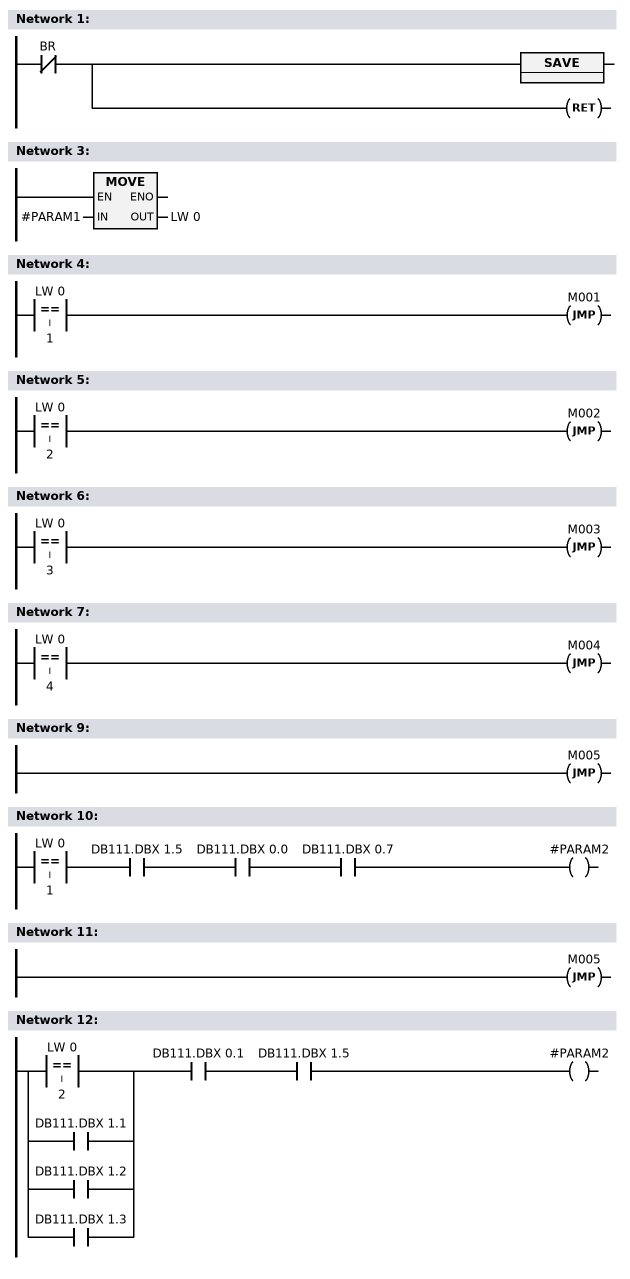
NETWORK
TITLE =
      AN    BR;
      SAVE;
      BEC;
NETWORK
TITLE =
      A     M 0.1;
      =     L 2.0;
NETWORK
TITLE =
      L     #PARAM1;
      T     LW 0;
      NOP   0;
NETWORK
TITLE =
      L     LW 0;
      L     1;
      ==I;
      JC    M001;
NETWORK
TITLE =
      L     LW 0;
      L     2;
      ==I;
      JC    M002;
NETWORK
TITLE =
      L     LW 0;
      L     3;
      ==I;
      JC    M003;
NETWORK
TITLE =
      L     LW 0;
      L     4;
      ==I;
      JC    M004;
NETWORK
TITLE =
      A     M 0.0;
      =     L 2.0;
NETWORK
TITLE =
      JU    M005;
NETWORK
TITLE =
M001: A(;
      L     LW 0;
      L     1;
      ==I;
      );
      A     DB111.DBX 1.5;
      A     DB111.DBX 0.0;
      A     DB111.DBX 0.7;
      =     #PARAM2;
NETWORK
TITLE =
      JU    M005;
NETWORK
TITLE =
M002: A(;
      O(;
      L     LW 0;
      L     2;
      ==I;
      );
      O     DB111.DBX 1.1;
      O     DB111.DBX 1.2;
      O     DB111.DBX 1.3;
      );
      A     DB111.DBX 0.1;
      A     DB111.DBX 1.5;
      =     #PARAM2;
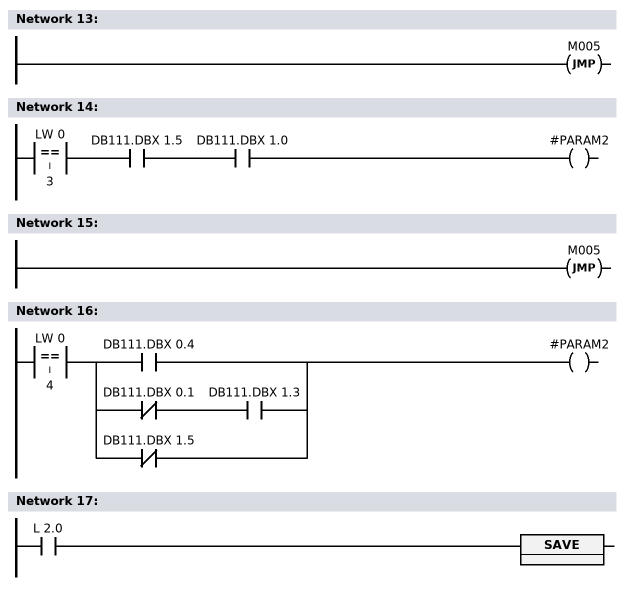
NETWORK
TITLE =
      JU    M005;
NETWORK
TITLE =
M003: A(;
      L     LW 0;
      L     3;
      ==I;
      );
      A     DB111.DBX 1.5;
      A     DB111.DBX 1.0;
      =     #PARAM2;
NETWORK
TITLE =
      JU    M005;
NETWORK
TITLE =
M004: A(;
      L     LW 0;
      L     4;
      ==I;
      );
      A(;
      O     DB111.DBX 0.4;
      O;
      AN    DB111.DBX 0.1;
      A     DB111.DBX 1.3;
      ON    DB111.DBX 1.5;
      );
      =     #PARAM2;
NETWORK
TITLE =
M005: A     L 2.0;
      SAVE;
END_FUNCTION

FUNCTION FC 93 : VOID
AUTHOR : A.Petz
VERSION : 0.2
BEGIN
// (block stored without names or comments; labels and parameter names are numbered)
NETWORK
TITLE =
      L     #PARAM1;
      DTB;
      T     LW 0;
NETWORK
TITLE =
      A     #PARAM2;
      JC    M002;
      L     LW 0;
      AW    W#16#FF;
      L     0;
      ==I;
      JC    M001;
      L     LW 0;
      AW    W#16#F;
      +     3;
      L     1000;
      *I;
      T     #PARAM3;
      L     LW 0;
      SRW   4;
      AW    W#16#F;
      SLW   2;
      +     2;
      L     1000;
      *I;
      T     #PARAM4;
      JU    M002;
M001: L     T#10M;
      T     #PARAM3;
      T     #PARAM4;
M002: NOP   0;
NETWORK
TITLE =
      AN    #PARAM2;
      JC    M004;
      L     LW 0;
      CAW;
      AW    W#16#FF;
      L     0;
      ==I;
      JC    M003;
      TAK;
      AW    W#16#F;
      +     3;
      L     1000;
      *I;
      T     #PARAM3;
      L     LW 0;
      SRW   12;
      AW    W#16#F;
      SLW   2;
      +     2;
      L     1000;
      *I;
      T     #PARAM4;
      JU    M004;
M003: L     T#10M;
      T     #PARAM3;
      T     #PARAM4;
M004: NOP   0;
END_FUNCTION

FUNCTION FC 94 : VOID
AUTHOR : SPAC_slh
FAMILY : GENERAL
NAME : General
VERSION : 1.0
BEGIN
// (block stored without names or comments; labels and parameter names are numbered)
NETWORK
TITLE =
      L     #PARAM1;
      T     LW 6;
      TAR1  LD 0;
      LAR1  P#L 4.0;
      L     B#16#0;
      T     LW 4;
      L     LW 6;
      AW    W#16#F;
      JZ    M001;
      +AR1;
      SET;
      S     L [AR1,P#0.0];
M001: LAR1  LD 0;
      L     LW 4;
      T     #PARAM2;
      L     LW 6;
      AW    W#16#FFF0;
      T     #PARAM3;
END_FUNCTION

FUNCTION FC 101 : VOID
AUTHOR : SPAC_slh
FAMILY : Diagnose
NAME : CK2OP
VERSION : 0.1
BEGIN
// (block stored without names or comments; labels and parameter names are numbered)
NETWORK
TITLE =
      TAR1  LD 10;
      TAR2  LD 14;
      L     P##PARAM1;
      LAR1;
      LAR2  P#L 0.0;
      L     W [AR1,P#0.0];
      T     LW [AR2,P#0.0];
      L     D [AR1,P#2.0];
      T     LD [AR2,P#2.0];
      L     D [AR1,P#6.0];
      T     LD [AR2,P#6.0];
      LAR1  LD 10;
      LAR2  LD 14;
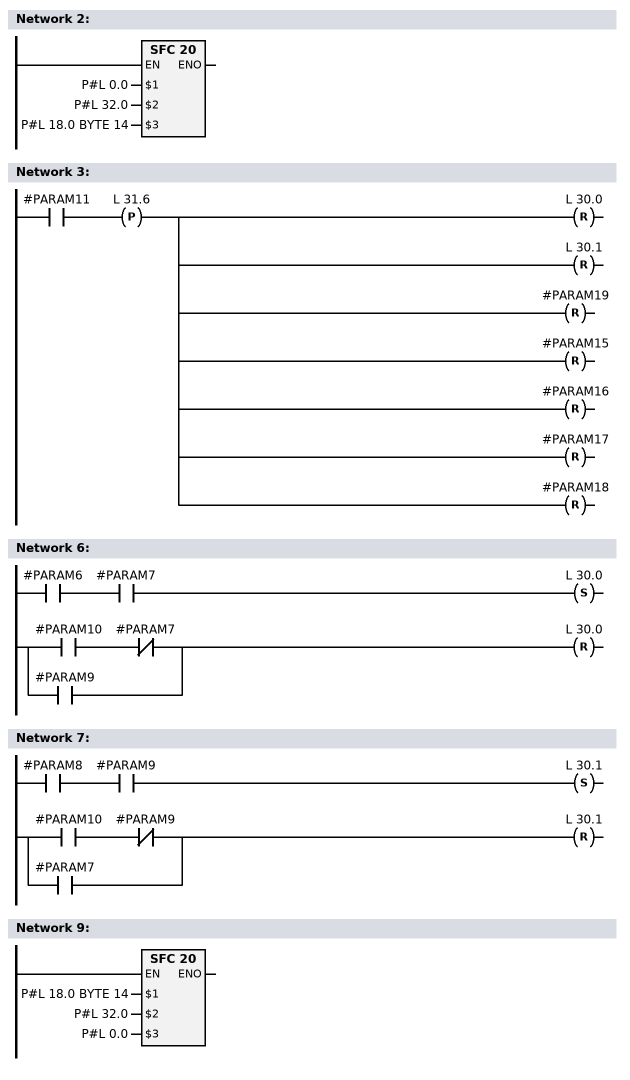
NETWORK
TITLE =
      CALL  SFC 20 (
           $1                       := P#L 0.0,
           $2                       := P#L 32.0,
           $3                       := P#L 18.0 BYTE 14);
      NOP   0;
NETWORK
TITLE =
      A     #PARAM11;
      FP    L 31.6;
      =     L 34.7;
      A     L 34.7;
      R     L 30.0;
      R     L 30.1;
      R     #PARAM19;
      R     #PARAM15;
      R     #PARAM16;
      R     #PARAM17;
      R     #PARAM18;
NETWORK
TITLE =
      L     T#0MS;
      L     #PARAM3;
      ==D;
      O     #PARAM12;
      JC    M004;
      R     L 34.3;
      A     #PARAM6;
      A     #PARAM8;
      AN    L 34.7;
      =     L 34.1;
      A     L 34.1;
      FP    L 31.0;
      =     L 34.2;
      AN    L 34.1;
      JC    M003;
      L     #PARAM2;
      AN    L 34.2;
      JC    M001;
      T     LD 18;
M001: L     LD 18;
      -D;
      JPZ   M002;
      L     L#2147483647;
      +D;
M002: L     #PARAM3;
      >=D;
      =     L 34.3;
M003: A     L 34.1;
      A     L 34.3;
      =     L 34.4;
      A     L 34.4;
      S     #PARAM19;
M004: NOP   0;
NETWORK
TITLE =
      A     #PARAM7;
      FP    L 31.4;
      =     L 34.5;
      A     #PARAM9;
      FP    L 31.5;
      =     L 34.6;
      L     T#0MS;
      L     #PARAM4;
      ==D;
      O     #PARAM13;
      JC    M008;
      R     L 34.3;
      A(;
      AN    #PARAM6;
      A     #PARAM7;
      AN    L 34.5;
      AN    L 30.0;
      O;
      AN    #PARAM8;
      A     #PARAM9;
      AN    L 34.6;
      AN    L 30.1;
      );
      AN    L 34.7;
      =     L 34.1;
      A     L 34.1;
      FP    L 31.1;
      =     L 34.2;
      AN    L 34.1;
      JC    M007;
      L     #PARAM2;
      AN    L 34.2;
      JC    M005;
      T     LD 22;
M005: L     LD 22;
      -D;
      JPZ   M006;
      L     L#2147483647;
      +D;
M006: L     #PARAM4;
      >=D;
      =     L 34.3;
M007: A     L 34.1;
      A     L 34.3;
      =     L 34.4;
      A     L 34.4;
      A     #PARAM7;
      S     #PARAM15;
      A     L 34.4;
      A     #PARAM9;
      S     #PARAM16;
M008: NOP   0;
NETWORK
TITLE =
      A     #PARAM6;
      A     #PARAM7;
      S     L 30.0;
      A(;
      A     #PARAM10;
      AN    #PARAM7;
      O     #PARAM9;
      );
      R     L 30.0;
      NOP   0;
NETWORK
TITLE =
      A     #PARAM8;
      A     #PARAM9;
      S     L 30.1;
      A(;
      A     #PARAM10;
      AN    #PARAM9;
      O     #PARAM7;
      );
      R     L 30.1;
      NOP   0;
NETWORK
TITLE =
      L     T#0MS;
      L     #PARAM5;
      ==D;
      O     #PARAM14;
      JC    M012;
      R     L 34.3;
      A(;
      A     L 30.0;
      AN    #PARAM6;
      O;
      A     L 30.1;
      AN    #PARAM8;
      );
      AN    L 34.7;
      =     L 34.1;
      A     L 34.1;
      FP    L 31.2;
      =     L 34.2;
      AN    L 34.1;
      JC    M011;
      L     #PARAM2;
      AN    L 34.2;
      JC    M009;
      T     LD 26;
M009: L     LD 26;
      -D;
      JPZ   M010;
      L     L#2147483647;
      +D;
M010: L     #PARAM5;
      >=D;
      =     L 34.3;
M011: A     L 34.1;
      A     L 34.3;
      =     L 34.4;
      A     L 34.4;
      A     L 30.0;
      AN    #PARAM6;
      S     #PARAM17;
      A     L 34.4;
      A     L 30.1;
      AN    #PARAM8;
      S     #PARAM18;
M012: NOP   0;
NETWORK
TITLE =
      CALL  SFC 20 (
           $1                       := P#L 18.0 BYTE 14,
           $2                       := P#L 32.0,
           $3                       := P#L 0.0);
      NOP   0;
END_FUNCTION

FUNCTION FC 102 : VOID
AUTHOR : SPAC_slh
FAMILY : Diagnose
NAME : CK1OP
VERSION : 0.1
BEGIN
// (block stored without names or comments; labels and parameter names are numbered)
NETWORK
TITLE =
      TAR1  LD 10;
      TAR2  LD 14;
      L     P##PARAM1;
      LAR1;
      LAR2  P#L 0.0;
      L     W [AR1,P#0.0];
      T     LW [AR2,P#0.0];
      L     D [AR1,P#2.0];
      T     LD [AR2,P#2.0];
      L     D [AR1,P#6.0];
      T     LD [AR2,P#6.0];
      LAR1  LD 10;
      LAR2  LD 14;
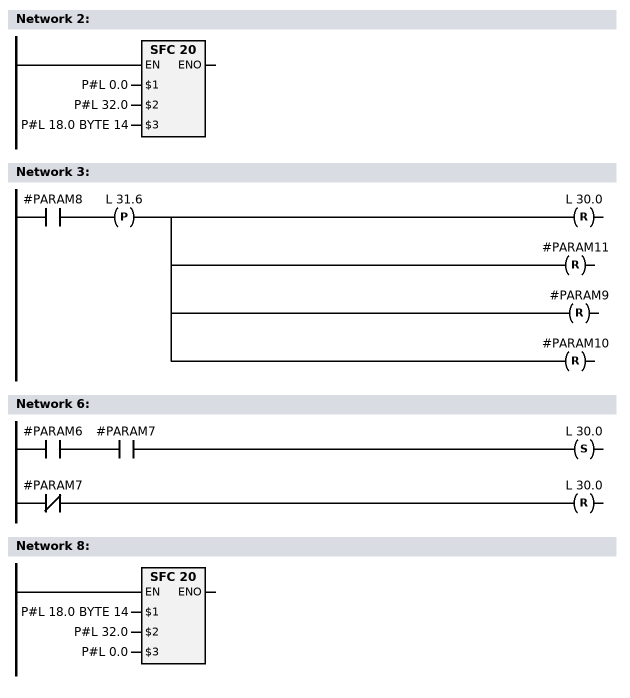
NETWORK
TITLE =
      CALL  SFC 20 (
           $1                       := P#L 0.0,
           $2                       := P#L 32.0,
           $3                       := P#L 18.0 BYTE 14);
      NOP   0;
NETWORK
TITLE =
      A     #PARAM8;
      FP    L 31.6;
      =     L 34.6;
      A     L 34.6;
      R     L 30.0;
      R     #PARAM11;
      R     #PARAM9;
      R     #PARAM10;
NETWORK
TITLE =
      L     T#0MS;
      L     #PARAM3;
      ==D;
      JC    M004;
      R     L 34.3;
      A     #PARAM6;
      AN    #PARAM7;
      AN    L 34.6;
      =     L 34.1;
      A     L 34.1;
      FP    L 31.0;
      =     L 34.2;
      AN    L 34.1;
      JC    M003;
      L     #PARAM2;
      AN    L 34.2;
      JC    M001;
      T     LD 18;
M001: L     LD 18;
      -D;
      JPZ   M002;
      L     L#2147483647;
      +D;
M002: L     #PARAM3;
      >=D;
      =     L 34.3;
M003: A     L 34.1;
      A     L 34.3;
      =     L 34.4;
      A     L 34.4;
      S     #PARAM11;
M004: NOP   0;
NETWORK
TITLE =
      A     #PARAM7;
      FP    L 31.4;
      =     L 34.5;
      L     T#0MS;
      L     #PARAM4;
      ==D;
      JC    M008;
      R     L 34.3;
      AN    #PARAM6;
      A     #PARAM7;
      AN    L 30.0;
      AN    L 34.6;
      =     L 34.1;
      A     L 34.1;
      FP    L 31.1;
      =     L 34.2;
      AN    L 34.1;
      JC    M007;
      L     #PARAM2;
      AN    L 34.2;
      JC    M005;
      T     LD 22;
M005: L     LD 22;
      -D;
      JPZ   M006;
      L     L#2147483647;
      +D;
M006: L     #PARAM4;
      >=D;
      =     L 34.3;
M007: A     L 34.1;
      A     L 34.3;
      =     L 34.4;
      A     L 34.4;
      S     #PARAM9;
M008: NOP   0;
NETWORK
TITLE =
      A     #PARAM6;
      A     #PARAM7;
      S     L 30.0;
      AN    #PARAM7;
      R     L 30.0;
      NOP   0;
NETWORK
TITLE =
      L     T#0MS;
      L     #PARAM5;
      ==D;
      JC    M012;
      R     L 34.3;
      A     L 30.0;
      AN    #PARAM6;
      AN    L 34.6;
      =     L 34.1;
      A     L 34.1;
      FP    L 31.2;
      =     L 34.2;
      AN    L 34.1;
      JC    M011;
      L     #PARAM2;
      AN    L 34.2;
      JC    M009;
      T     LD 26;
M009: L     LD 26;
      -D;
      JPZ   M010;
      L     L#2147483647;
      +D;
M010: L     #PARAM5;
      >=D;
      =     L 34.3;
M011: A     L 34.1;
      A     L 34.3;
      =     L 34.4;
      A     L 34.4;
      A     L 30.0;
      AN    #PARAM6;
      S     #PARAM10;
M012: NOP   0;
NETWORK
TITLE =
      CALL  SFC 20 (
           $1                       := P#L 18.0 BYTE 14,
           $2                       := P#L 32.0,
           $3                       := P#L 0.0);
      NOP   0;
END_FUNCTION

FUNCTION FC 111 : VOID
AUTHOR : APetz
VERSION : 0.1
BEGIN
// (block stored without names or comments; labels and parameter names are numbered)
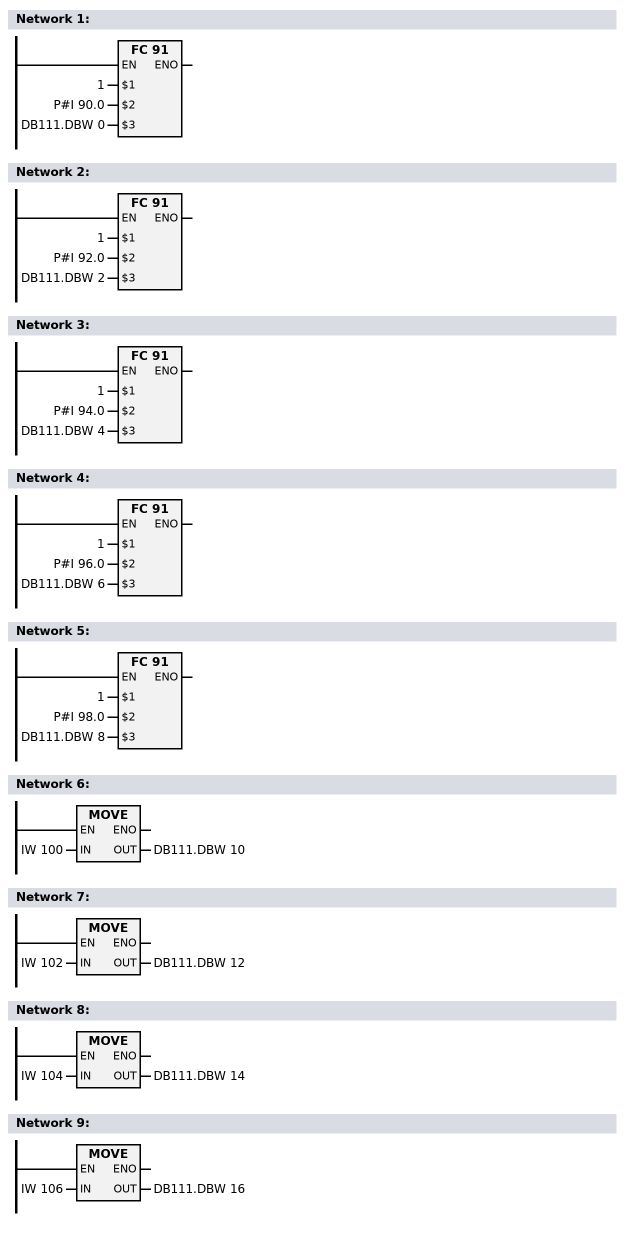
NETWORK
TITLE =
      CALL  FC 91 (
           $1                       := 1,
           $2                       := P#I 90.0,
           $3                       := DB111.DBW 0);
      NOP   0;
NETWORK
TITLE =
      CALL  FC 91 (
           $1                       := 1,
           $2                       := P#I 92.0,
           $3                       := DB111.DBW 2);
      NOP   0;
NETWORK
TITLE =
      CALL  FC 91 (
           $1                       := 1,
           $2                       := P#I 94.0,
           $3                       := DB111.DBW 4);
      NOP   0;
NETWORK
TITLE =
      CALL  FC 91 (
           $1                       := 1,
           $2                       := P#I 96.0,
           $3                       := DB111.DBW 6);
      NOP   0;
NETWORK
TITLE =
      CALL  FC 91 (
           $1                       := 1,
           $2                       := P#I 98.0,
           $3                       := DB111.DBW 8);
      NOP   0;
NETWORK
TITLE =
      L     IW 100;
      T     DB111.DBW 10;
      NOP   0;
NETWORK
TITLE =
      L     IW 102;
      T     DB111.DBW 12;
      NOP   0;
NETWORK
TITLE =
      L     IW 104;
      T     DB111.DBW 14;
      NOP   0;
NETWORK
TITLE =
      L     IW 106;
      T     DB111.DBW 16;
      NOP   0;
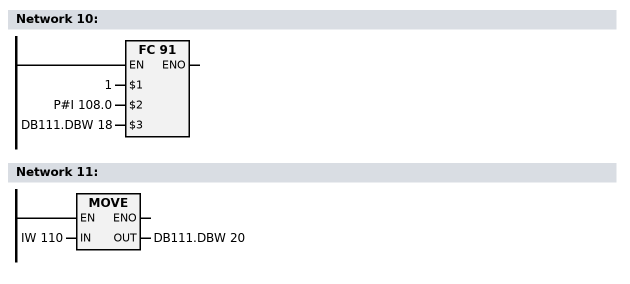
NETWORK
TITLE =
      CALL  FC 91 (
           $1                       := 1,
           $2                       := P#I 108.0,
           $3                       := DB111.DBW 18);
      NOP   0;
NETWORK
TITLE =
      L     IW 110;
      T     DB111.DBW 20;
      NOP   0;
END_FUNCTION

FUNCTION FC 112 : VOID
AUTHOR : APetz
VERSION : 0.1
BEGIN
// (block stored without names or comments; labels and parameter names are numbered)
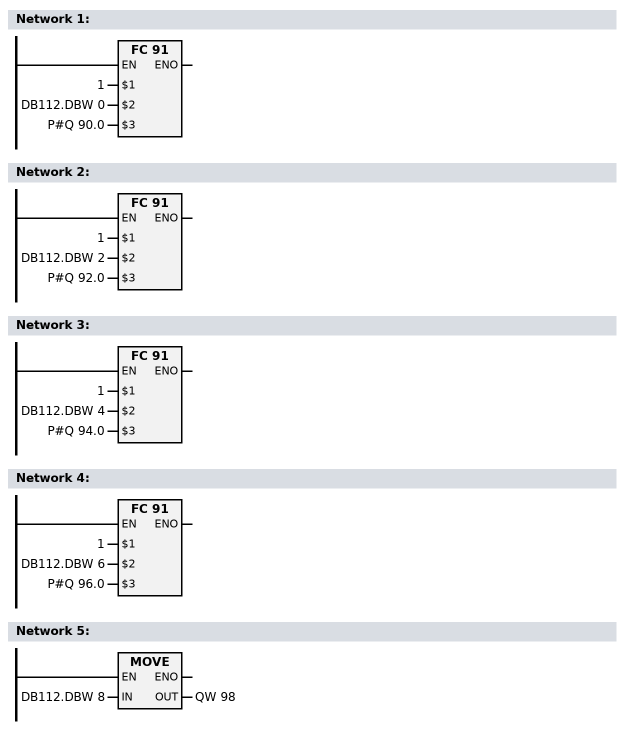
NETWORK
TITLE =
      CALL  FC 91 (
           $1                       := 1,
           $2                       := DB112.DBW 0,
           $3                       := P#Q 90.0);
      NOP   0;
NETWORK
TITLE =
      CALL  FC 91 (
           $1                       := 1,
           $2                       := DB112.DBW 2,
           $3                       := P#Q 92.0);
      NOP   0;
NETWORK
TITLE =
      CALL  FC 91 (
           $1                       := 1,
           $2                       := DB112.DBW 4,
           $3                       := P#Q 94.0);
      NOP   0;
NETWORK
TITLE =
      CALL  FC 91 (
           $1                       := 1,
           $2                       := DB112.DBW 6,
           $3                       := P#Q 96.0);
      NOP   0;
NETWORK
TITLE =
      L     DB112.DBW 8;
      T     QW 98;
      NOP   0;
END_FUNCTION

FUNCTION FC 120 : VOID
AUTHOR : APetz
FAMILY : AUTOMAT
NAME : SusDoor
VERSION : 1.0
BEGIN
// (block stored without names or comments; labels and parameter names are numbered)
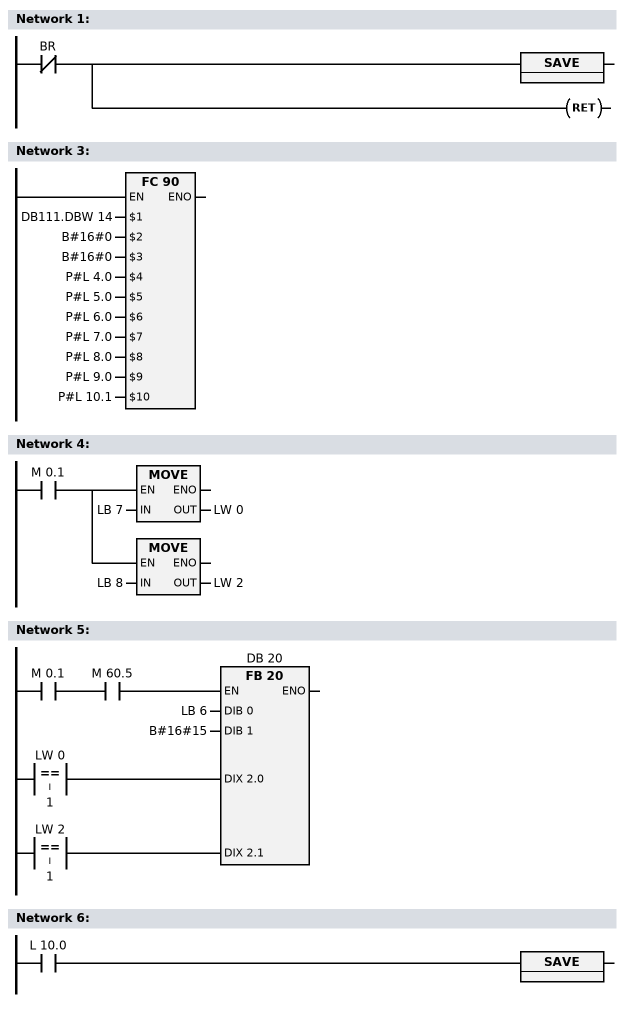
NETWORK
TITLE =
      AN    BR;
      SAVE;
      BEC;
NETWORK
TITLE =
      A     M 0.1;
      =     L 10.0;
NETWORK
TITLE =
      CALL  FC 90 (
           $1                       := DB111.DBW 14,
           $2                       := B#16#0,
           $3                       := B#16#0,
           $4                       := P#L 4.0,
           $5                       := P#L 5.0,
           $6                       := P#L 6.0,
           $7                       := P#L 7.0,
           $8                       := P#L 8.0,
           $9                       := P#L 9.0,
           $10                      := P#L 10.1);
      NOP   0;
NETWORK
TITLE =
      A     M 0.1;
      =     L 11.0;
      A     L 11.0;
      JNB   M001;
      L     LB 7;
      T     LW 0;
M001: NOP   0;
      A     L 11.0;
      JNB   M002;
      L     LB 8;
      T     LW 2;
M002: NOP   0;
NETWORK
TITLE =
      A(;
      L     LW 0;
      L     1;
      ==I;
      );
      =     L 11.0;
      BLD   103;
      A(;
      L     LW 2;
      L     1;
      ==I;
      );
      =     L 11.1;
      BLD   103;
      A     M 0.1;
      A     M 60.5;
      JNB   M003;
      CALL  FB 20 , DB 20 (
           DIB 0                    := LB 6,
           DIB 1                    := B#16#15,
           DIX 2.0                  := L 11.0,
           DIX 2.1                  := L 11.1);
M003: NOP   0;
NETWORK
TITLE =
      A     L 10.0;
      SAVE;
END_FUNCTION

FUNCTION FC 121 : VOID
AUTHOR : APetz
VERSION : 0.1
BEGIN
// (block stored without names or comments; labels and parameter names are numbered)
NETWORK
TITLE =
      AN    BR;
      SAVE;
      BEC;
NETWORK
TITLE =
      A     M 0.1;
      =     L 0.0;
NETWORK
TITLE =
      A     I 2.0;
      =     M 128.6;
      A     I 2.1;
      =     M 128.7;
      A     I 2.2;
      =     M 129.0;
      A     I 2.3;
      =     M 129.1;
      A     I 3.0;
      =     M 129.2;
      A     I 3.1;
      =     M 129.3;
      A     I 3.2;
      =     M 129.4;
      A     I 4.0;
      =     M 129.5;
      A     I 4.1;
      =     M 129.6;
      A     I 4.2;
      =     M 129.7;
      A     I 4.3;
      =     M 130.0;
NETWORK
TITLE =
      A     L 0.0;
      SAVE;
END_FUNCTION

FUNCTION FC 122 : VOID
AUTHOR : APetz
VERSION : 0.1
BEGIN
// (block stored without names or comments; labels and parameter names are numbered)
NETWORK
TITLE =
      AN    BR;
      SAVE;
      BEC;
NETWORK
TITLE =
      A     M 0.1;
      =     L 0.0;
NETWORK
TITLE =
      A     M 195.4;
      =     Q 6.0;
      A     M 195.5;
      =     Q 6.1;
      A     M 195.6;
      =     Q 6.2;
NETWORK
TITLE =
      A     L 0.0;
      SAVE;
END_FUNCTION

DATA_BLOCK DB 2
AUTHOR : SPAC_slh
VERSION : 0.1
UDT 2
BEGIN
END_DATA_BLOCK

DATA_BLOCK DB 20
AUTHOR : SPAC_slh
FAMILY : AUTOMAT
VERSION : 0.0
FB 20
BEGIN
END_DATA_BLOCK

DATA_BLOCK DB 100
AUTHOR : SPAC_slh
VERSION : 0.0
FB 100
BEGIN
END_DATA_BLOCK

DATA_BLOCK DB 101
VERSION : 0.1
UDT 101
BEGIN
END_DATA_BLOCK

DATA_BLOCK DB 111
AUTHOR : M.Kögel
VERSION : 0.1
BEGIN
// 26 bytes; values not shown
END_DATA_BLOCK

DATA_BLOCK DB 112
AUTHOR : APetz
VERSION : 0.1
BEGIN
// 12 bytes; values not shown
END_DATA_BLOCK

ORGANIZATION_BLOCK OB 1
AUTHOR : APetz
VERSION : 0.1
BEGIN
// (block stored without names or comments; labels and parameter names are numbered)
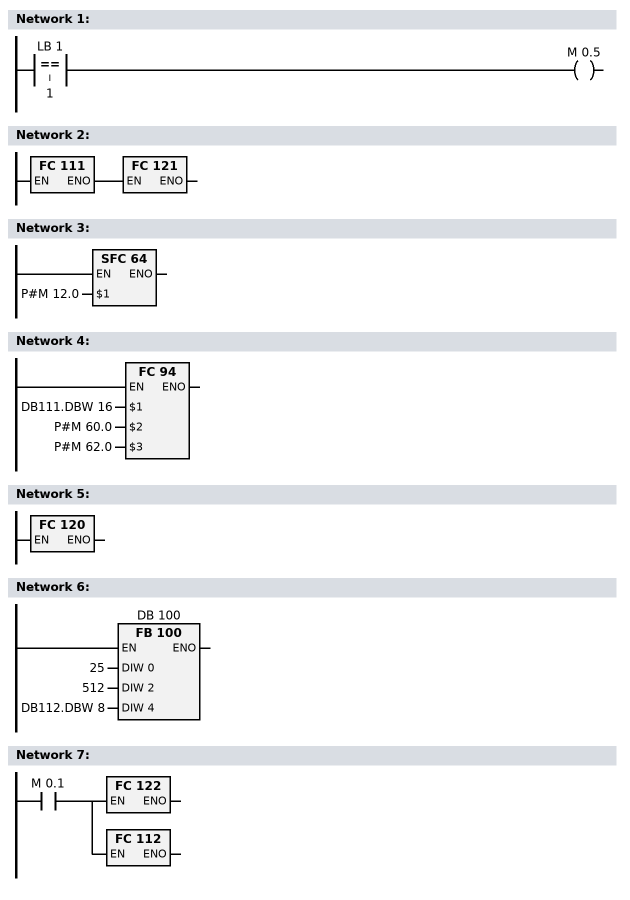
NETWORK
TITLE =
      L     LB 1;
      L     1;
      ==I;
      =     M 0.5;
NETWORK
TITLE =
      A(;
      CALL  FC 111;
      A     BR;
      );
      JNB   M001;
      CALL  FC 121;
M001: NOP   0;
NETWORK
TITLE =
      CALL  SFC 64 (
           $1                       := P#M 12.0);
      NOP   0;
NETWORK
TITLE =
      CALL  FC 94 (
           $1                       := DB111.DBW 16,
           $2                       := P#M 60.0,
           $3                       := P#M 62.0);
      NOP   0;
NETWORK
TITLE =
      CALL  FC 120;
      NOP   0;
NETWORK
TITLE =
      CALL  FB 100 , DB 100 (
           DIW 0                    := 25,
           DIW 2                    := 512,
           DIW 4                    := DB112.DBW 8);
      NOP   0;
NETWORK
TITLE =
      A     M 0.1;
      =     L 20.0;
      A     L 20.0;
      JNB   M002;
      CALL  FC 122;
M002: NOP   0;
      A     L 20.0;
      JNB   M003;
      CALL  FC 112;
M003: NOP   0;
END_ORGANIZATION_BLOCK

ORGANIZATION_BLOCK OB 82
VERSION : 0.1
BEGIN
// (block stored without names or comments; labels and parameter names are numbered)
NETWORK
TITLE =
END_ORGANIZATION_BLOCK

ORGANIZATION_BLOCK OB 85
VERSION : 0.1
BEGIN
// (block stored without names or comments; labels and parameter names are numbered)
NETWORK
TITLE =
END_ORGANIZATION_BLOCK

ORGANIZATION_BLOCK OB 86
VERSION : 0.1
BEGIN
// (block stored without names or comments; labels and parameter names are numbered)
NETWORK
TITLE =
END_ORGANIZATION_BLOCK

ORGANIZATION_BLOCK OB 100
VERSION : 0.1
BEGIN
// (block stored without names or comments; labels and parameter names are numbered)
NETWORK
TITLE =
      SET;
      R     M 0.0;
      S     M 0.1;
      S     M 0.6;
END_ORGANIZATION_BLOCK

ORGANIZATION_BLOCK OB 121
VERSION : 0.1
BEGIN
// (block stored without names or comments; labels and parameter names are numbered)
END_ORGANIZATION_BLOCK

ORGANIZATION_BLOCK OB 122
VERSION : 0.1
BEGIN
// (block stored without names or comments; labels and parameter names are numbered)
END_ORGANIZATION_BLOCK

